(* IEC 61131-3 sources: cstr_project/plc/appdata/st_files, 3 files *)

(* ---- 877151.st ---- *)
PROGRAM cstr_control
  VAR
    T_reactor AT %IW100 : INT;
    Ca_reactor AT %IW101 : INT;
    q_setpoint AT %QW2 : INT;
    Caf_setpoint AT %QW3 : INT;
    Tc_setpoint AT %QW4 : INT;
    T_high_alarm AT %QX0.0 : BOOL := FALSE;
    manual_mode AT %IX0.0 : BOOL := TRUE;
  END_VAR
  VAR
    relay1 AT %QX0.1 : BOOL := FALSE;
    relay2 AT %QX0.2 : BOOL := TRUE;
  END_VAR

  q_setpoint := 10000;
  Caf_setpoint := 1000;

  IF manual_mode = TRUE THEN
    Tc_setpoint := 30000;
    T_high_alarm := FALSE;
  ELSE
    Tc_setpoint := 29000;
    T_high_alarm := TRUE;
  END_IF;

END_PROGRAM

CONFIGURATION Config0

  RESOURCE Res0 ON PLC
    TASK task0(INTERVAL := T#20ms,PRIORITY := 0);
    PROGRAM instance0 WITH task0 : cstr_control;
  END_RESOURCE
END_CONFIGURATION

(* ---- blank_program.st ---- *)
PROGRAM prog0
  VAR
    var_in : BOOL;
    var_out : BOOL;
  END_VAR

  var_out := var_in;
END_PROGRAM

CONFIGURATION Config0

  RESOURCE Res0 ON PLC
    TASK Main(INTERVAL := T#50ms,PRIORITY := 0);
    PROGRAM Inst0 WITH Main : prog0;
  END_RESOURCE
END_CONFIGURATION

(* ---- cstr_control.st ---- *)
PROGRAM cstr_control
  VAR
    T_reactor AT %IW0 : INT;
    Ca_reactor AT %IW2 : INT;
    q_setpoint AT %QW4 : INT;
    Caf_setpoint AT %QW6 : INT;
    Tc_setpoint AT %QW8 : INT;
    T_high_alarm AT %QX0.0 : BOOL := FALSE;
    manual_mode AT %IX0.0 : BOOL := TRUE;
  END_VAR

  q_setpoint := 10000;
  Caf_setpoint := 1000;

  IF manual_mode = TRUE THEN
    Tc_setpoint := 30000;
    T_high_alarm := FALSE;
  ELSE
    Tc_setpoint := 29000;
    T_high_alarm := TRUE;
  END_IF;

END_PROGRAM

CONFIGURATION Config0

  RESOURCE Res0 ON PLC
    TASK task0(INTERVAL := T#100ms,PRIORITY := 0);
    PROGRAM instance0 WITH task0 : cstr_control;
  END_RESOURCE
END_CONFIGURATION
